FUNCTION_BLOCK FB_Operate
VAR_INPUT
	i_nOperation : E_Op := E_Op.NONE; // Select which operation to run, if any
	i_bCancel : BOOL; // Flag to cancel the current operation
END_VAR
VAR_OUTPUT
	q_bBusy : BOOL := FALSE; // Flag for if an operation is running
	q_nOperation : E_Op := E_Op.NONE; // Operation that is currently running
END_VAR
VAR
	(* Operations *)
	fbPumpTransportTube : FB_PumpTransportTube;
	fbVentTransportTube : FB_VentTransportTube;
	fbPumpSwitchbox : FB_PumpSwitchbox;
	fbSlowPumpSwitchbox : FB_SlowPumpSwitchbox;
	fbVentPumpStation : FB_VentPumpStation;
	fbVentSwitchbox : FB_VentSwitchbox;
	fbSlowVentSwitchbox : FB_SlowVentSwitchbox;
END_VAR

(* Run operations, but don't start any new operations if another operation is still running *)

// If there isn't a currently running operation, then the input operation will become the new running operation
// Also, don't switch the operation as long as another operation is still busy!
IF NOT q_bBusy THEN
	q_nOperation := i_nOperation;
END_IF

// Start execution of selected operation. Other operations will idle
fbPumpTransportTube(
	i_bExecute := q_nOperation = E_Op.POT1, 
	i_bCancel := i_bCancel,
	i_eTransportTube := E_TransportTube.BI1
);
q_bBusy := q_bBusy OR fbPumpTransportTube.q_bBusy;

fbVentTransportTube(
	i_bExecute := q_nOperation = E_Op.VOT1,
	i_bCancel := i_bCancel,
	i_eTransportTube := E_TransportTube.BI1
);

fbPumpSwitchbox(i_bExecute := q_nOperation = E_Op.PSB,
	i_bCancel := i_bCancel);
q_bBusy := q_bBusy OR fbPumpSwitchbox.q_bBusy;

fbSlowPumpSwitchbox(i_bExecute := q_nOperation = E_Op.SPSB,
	i_bCancel := i_bCancel);
q_bBusy := q_bBusy OR fbSlowPumpSwitchbox.q_bBusy;	
	
fbVentPumpStation(i_bExecute := q_nOperation = E_Op.VPS,
	i_bCancel := i_bCancel);
q_bBusy := q_bBusy OR fbVentPumpStation.q_bBusy;	
	
fbVentSwitchbox(i_bExecute := q_nOperation = E_Op.VSB,
	i_bCancel := i_bCancel);
q_bBusy := q_bBusy OR fbVentSwitchbox.q_bBusy;

fbVentSwitchbox(i_bExecute := q_nOperation = E_Op.SVSB,
	i_bCancel := i_bCancel);
q_bBusy := q_bBusy OR fbSlowVentSwitchbox.q_bBusy;

// If there isn't an operation running, then set opertion to none
IF NOT q_bBusy THEN
	q_nOperation := E_Op.NONE;
END_IF

END_FUNCTION_BLOCK

(* stored: Version 1.1.0.1, ProductVersion 3.1.4024.0
   POU FB_Operate: Id {8ee47251-2ac9-09b7-2785-97e47b267431}, SpecialFunc None *)
